FUNCTION_BLOCK IntComparator IMPLEMENTS I_Comparator,I_StepCondition
VAR_INPUT
END_VAR
VAR_OUTPUT
END_VAR
VAR
	uiSelector 		: UINT;
	rInternTarget1 	: REFERENCE TO INT;
	rInternTarget2 	: REFERENCE TO INT;
	bValue			: BOOL;
END_VAR

IF NOT __ISVALIDREF( rInternTarget1 )
OR NOT __ISVALIDREF( rInternTarget1 )
THEN
	uiSelector := 0;
END_IF 

CASE uiSelector OF

	0:;
		
	10:
		bValue := mEquals(rInternTarget1,rInternTarget2);
		
	20:
		bValue := mGreaterThan(rInternTarget1,rInternTarget2);
	
	30:
		bValue := mLessThan(rInternTarget1,rInternTarget2);
	
	40:
		bValue := mGreaterEquals(rInternTarget1,rInternTarget2);
		
	50:
		bValue := mLessEquals(rInternTarget1,rInternTarget2);
		
END_CASE

{warning 'Eigenschaftenimplementierung hinzufügen'}
PROPERTY getValue : BOOL
GET
getValue := bValue;
END_GET
END_PROPERTY

METHOD mEquals : BOOL;
VAR_INPUT
	rTarget1 : REFERENCE TO INT;
	rTarget2 : REFERENCE TO INT;
END_VAR
uiSelector := 10;
rInternTarget1 REF= rTarget1;
rInternTarget2 REF= rTarget2;

mEquals := ( rTarget1 = rTarget2 );
END_METHOD

METHOD PUBLIC mGreaterEquals : BOOL
VAR_INPUT
	rTarget1 : REFERENCE TO INT;
	rTarget2 : REFERENCE TO INT;
END_VAR
uiSelector := 40;
rInternTarget1 REF= rTarget1;
rInternTarget2 REF= rTarget2;

mGreaterEquals := ( rTarget1 >= rTarget2 );
END_METHOD

METHOD mGreaterThan : BOOL;
VAR_INPUT
	rTarget1 : REFERENCE TO INT;
	rTarget2 : REFERENCE TO INT;
END_VAR
uiSelector := 20;
rInternTarget1 REF= rTarget1;
rInternTarget2 REF= rTarget2;

mGreaterThan := ( rTarget1 >= rTarget2 );
END_METHOD

METHOD mLessEquals : BOOL
VAR_INPUT
	rTarget1 : REFERENCE TO INT;
	rTarget2 : REFERENCE TO INT;
END_VAR
uiSelector := 50;
rInternTarget1 REF= rTarget1;
rInternTarget2 REF= rTarget2;

mLessEquals := ( rTarget1 <= rTarget2 );
END_METHOD

METHOD mLessThan : BOOL;
VAR_INPUT
	rTarget1 : REFERENCE TO INT;
	rTarget2 : REFERENCE TO INT;
END_VAR
uiSelector := 30;
rInternTarget1 REF= rTarget1;
rInternTarget2 REF= rTarget2;

mLessThan := ( rTarget1 < rTarget2 );
END_METHOD

{warning 'Eigenschaftenimplementierung hinzufügen'}
PROPERTY setValue : BOOL
SET
bValue := setValue;
END_SET
END_PROPERTY

END_FUNCTION_BLOCK

(* stored: Version 1.1.0.1, ProductVersion 3.1.4024.0
   POU IntComparator: Id {3887696e-249c-4127-a9b7-24cc2c49dd21}, SpecialFunc None
   Property getValue: Id {afd56121-700d-4014-bca2-5bb07b48e610}
   Get Get: Id {ae278716-3830-48b7-bb04-303bb67d064a}
   Method mEquals: Id {ecbde6ca-eb5d-4d58-80c9-be4a96afd96a}
   Method mGreaterEquals: Id {4452399b-046f-4ee3-9af7-6d8a41149e66}
   Method mGreaterThan: Id {3d1d9bc7-3a4d-4ab4-8364-381aefd184db}
   Method mLessEquals: Id {efe1a045-e16a-43a8-9cb8-1e9a363bd6c0}
   Method mLessThan: Id {96bd4fbe-6997-4fb4-ac48-3132e1d504cb}
   Property setValue: Id {5bc06297-4e2e-4be4-a470-f1b8a8292168}
   Set Set: Id {3df1d4ae-6d89-4fba-9c6f-4ad0b56a7b0f} *)
